(* IEC 61131-3 sources: plc-ics/PumpStation (ST), 2 files *)

(* ---- PumpController.st ---- *)
FUNCTION_BLOCK PumpController
VAR_INPUT
    StartCmd    : BOOL;
    StopCmd     : BOOL;
    DryRun      : BOOL;
    Overheat    : BOOL;
    AutoMode    : BOOL;
    MinLevel    : BOOL;
    MaxLevel    : BOOL;
END_VAR

VAR_OUTPUT
    PumpOn      : BOOL;
    Alarm       : BOOL;
END_VAR

VAR
    DelayStart  : TON;
END_VAR

// Таймер на 5 секунд задержки запуска
DelayStart(IN := StartCmd AND NOT PumpOn, PT := T#5s);

IF StopCmd THEN
    PumpOn := FALSE;
    Alarm := FALSE;

ELSIF Overheat OR DryRun THEN
    Alarm := TRUE;
    PumpOn := FALSE;

ELSIF AutoMode THEN
    IF NOT MaxLevel AND MinLevel AND DelayStart.Q THEN
        PumpOn := TRUE;
    ELSE
        PumpOn := FALSE;
    END_IF;

ELSE // Ручной режим
    IF StartCmd AND NOT Overheat AND NOT DryRun THEN
        PumpOn := TRUE;
    END_IF;
END_IF;

(* ---- main.st ---- *)
PROGRAM MAIN
VAR
    Pump1  : PumpController;
    Pump2  : PumpController;
    Toggle : BOOL := FALSE;
    TimerToggle : TON;
END_VAR

// Переключатель режимов
IF GlobalVars.StartAuto THEN
    GlobalVars.ModeAuto := TRUE;
ELSIF GlobalVars.StartManual THEN
    GlobalVars.ModeAuto := FALSE;
END_IF;

// Таймер переключения насосов каждые 60 секунд
TimerToggle(IN := TRUE, PT := T#60s);
IF TimerToggle.Q THEN
    Toggle := NOT Toggle;
    TimerToggle(IN := FALSE); // Сброс
    TimerToggle(IN := TRUE);  // Переустановка
END_IF;

IF GlobalVars.ModeAuto THEN
    GlobalVars.CurrentModeText := 'Автоматический';
ELSE
    GlobalVars.CurrentModeText := 'Ручной';
END_IF;

// Ручной режим
IF NOT GlobalVars.ModeAuto THEN
    Pump1(
        StartCmd := GlobalVars.ManualPump1,
        StopCmd := GlobalVars.StopButton,
        DryRun := GlobalVars.DryRunSensor,
        Overheat := GlobalVars.OverheatPump1,
        AutoMode := FALSE,
        MinLevel := GlobalVars.LowLevel,
        MaxLevel := GlobalVars.HighLevel
    );

    Pump2(
        StartCmd := GlobalVars.ManualPump2,
        StopCmd := GlobalVars.StopButton,
        DryRun := GlobalVars.DryRunSensor,
        Overheat := GlobalVars.OverheatPump2,
        AutoMode := FALSE,
        MinLevel := GlobalVars.LowLevel,
        MaxLevel := GlobalVars.HighLevel
    );

ELSE
    // Автоматический режим с чередованием
    IF Toggle THEN
        Pump1(
            StartCmd := TRUE,
            StopCmd := GlobalVars.StopButton,
            DryRun := GlobalVars.DryRunSensor,
            Overheat := GlobalVars.OverheatPump1,
            AutoMode := TRUE,
            MinLevel := GlobalVars.LowLevel,
            MaxLevel := GlobalVars.HighLevel
        );

        Pump2(
            StartCmd := FALSE,
            StopCmd := GlobalVars.StopButton,
            DryRun := GlobalVars.DryRunSensor,
            Overheat := GlobalVars.OverheatPump2,
            AutoMode := TRUE,
            MinLevel := GlobalVars.LowLevel,
            MaxLevel := GlobalVars.HighLevel
        );
    ELSE
        Pump1(
            StartCmd := FALSE,
            StopCmd := GlobalVars.StopButton,
            DryRun := GlobalVars.DryRunSensor,
            Overheat := GlobalVars.OverheatPump1,
            AutoMode := TRUE,
            MinLevel := GlobalVars.LowLevel,
            MaxLevel := GlobalVars.HighLevel
        );

        Pump2(
            StartCmd := TRUE,
            StopCmd := GlobalVars.StopButton,
            DryRun := GlobalVars.DryRunSensor,
            Overheat := GlobalVars.OverheatPump2,
            AutoMode := TRUE,
            MinLevel := GlobalVars.LowLevel,
            MaxLevel := GlobalVars.HighLevel
        );
    END_IF;
END_IF;

// Вывод статусов насосов
GlobalVars.Pump1Status := Pump1.PumpOn;
GlobalVars.Pump2Status := Pump2.PumpOn;
